// TIA Portal V16 export
// export: Created 2021-09-08T12:46:14.6503974Z, ExportSetting WithDefaults, DisplayName Totally Integrated Automation Portal, DisplayVersion V16 Update 3, DisplayName TIA Portal Version Control Interface, DisplayVersion V16 Update 2, DisplayName TIA Portal Openness, DisplayVersion V16 Update 3, DisplayName TIA Portal Teamcenter Gateway, DisplayVersion V16, DisplayName STEP 7 Professional, DisplayVersion V16 Update 3, DisplayName STEP 7 Safety, DisplayVersion V16, DisplayName WinCC Advanced, DisplayVersion V16 Update 3
DATA_BLOCK "dtUF"   // DB23
{ S7_Optimized_Access := 'FALSE' }
VERSION : 0.1
// stored: AutoNumber true, DBAccessibleFromOPCUA true, IsOnlyStoredInLoadMemory false, IsWriteProtectedInAS false
   VAR RETAIN
      modeUF1 : Bool;
      modeUF2 : Bool;
      cmAuto : Bool;
      flagUF1 : "UF_FLAGS";
      flagUF2 { S7_SetPoint := 'True'} : "UF_FLAGS";
      bUF1 { S7_SetPoint := 'True'} : "UF_COMMANDS";
      bUF2 { S7_SetPoint := 'True'} : "UF_COMMANDS";
      countersUF1 { S7_SetPoint := 'True'} : "UF_COUNTERS";
      countersUF2 { S7_SetPoint := 'True'} : "UF_COUNTERS";
      parUF1 : "UF_PARAMETRS";
      parUF2 { S7_SetPoint := 'True'} : "UF_PARAMETRS";
   END_VAR
BEGIN
END_DATA_BLOCK
